FUNCTION_BLOCK CloseValve
VAR_INPUT
END_VAR
VAR_OUTPUT
	closeValve : BOOL := FALSE;
END_VAR
VAR
	readyToClose : BOOL := FALSE;
END_VAR

IF GVL.sensorN1 AND GVL.sensorN2 THEN
	closeValve := TRUE;
	readyToClose := TRUE;
ELSIF NOT GVL.sensorN1 AND NOT GVL.sensorN2 THEN
	closeValve := FALSE;
END_IF

IF NOT GVL.sensorN1 AND GVL.sensorN2 AND NOT readyToClose THEN 
	CloseValve := TRUE;
END_IF

END_FUNCTION_BLOCK

(* stored: Version 1.1.0.1, ProductVersion 3.1.4024.13
   POU CloseValve: Id {dccdc7eb-8f11-48b0-ba86-f0c95f914d23}, SpecialFunc None *)
